Xinje XCPPro project, PLC1: XC2-32 (software 3.3L)

PROGRAM Ladder

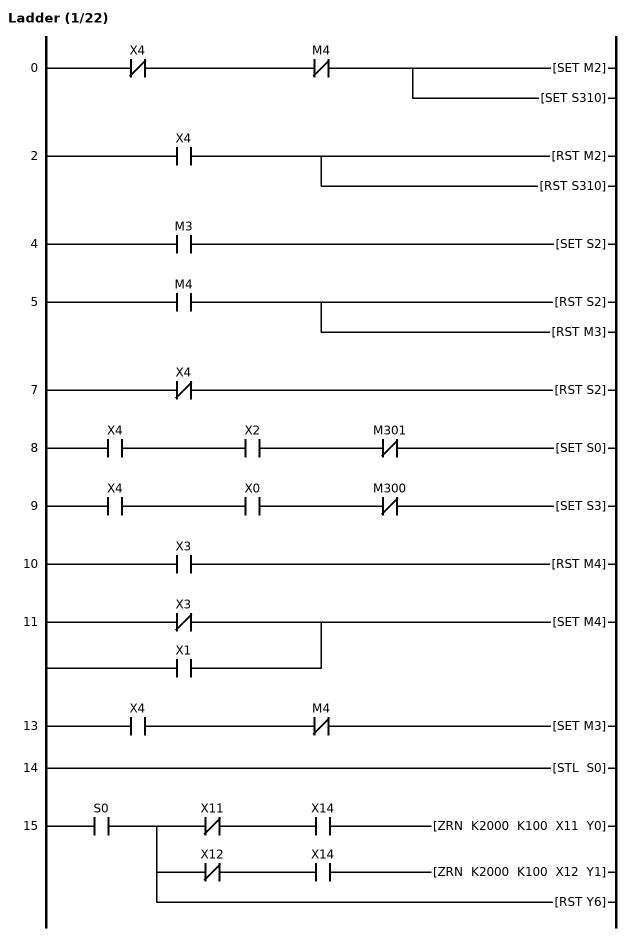
LDI    X4
ANI    M4
SET    M2
SET    S310
LD     X4
RST    M2
RST    S310
LD     M3
SET    S2
LD     M4
RST    S2
RST    M3
LDI    X4
RST    S2
LD     X4
AND    X2
ANI    M301
SET    S0
LD     X4
AND    X0
ANI    M300
SET    S3
LD     X3
RST    M4
LDI    X3
OR     X1
SET    M4
LD     X4
ANI    M4
SET    M3
STL    S0
LD     S0
MPS
ANI    X11
AND    X14
ZRN    K2000 K100 X11 Y0
MRD
ANI    X12
AND    X14
ZRN    K2000 K100 X12 Y1
MPP
RST    Y6

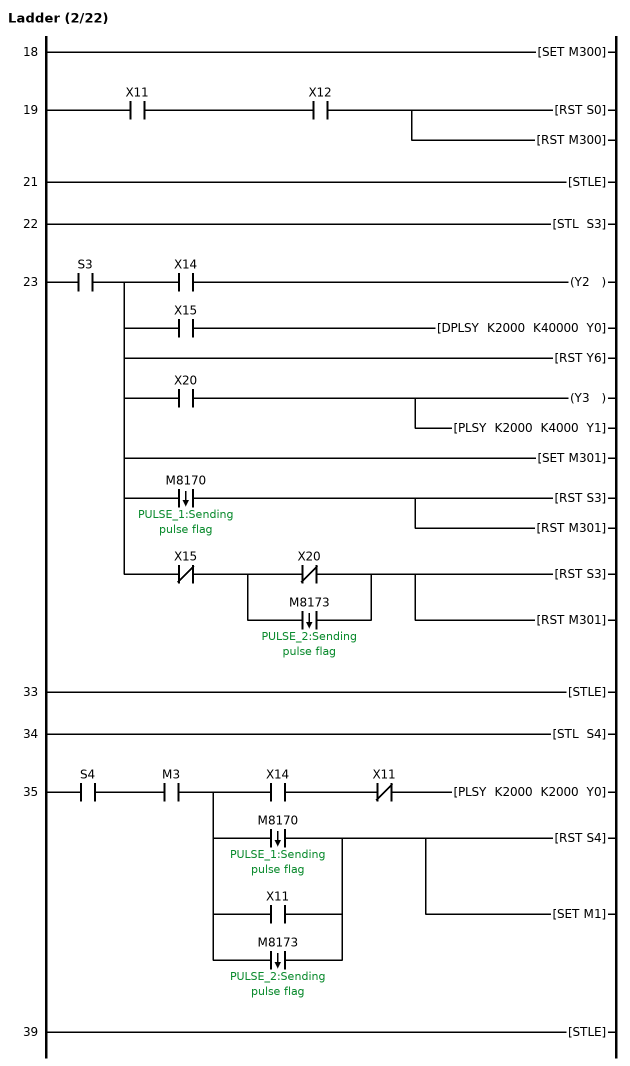
SET    M300
LD     X11
AND    X12
RST    S0
RST    M300
STLE
STL    S3
LD     S3
MPS
AND    X14
OUT    Y2
MRD
AND    X15
DPLSY  K2000 K40000 Y0
MRD
RST    Y6
AND    X20
OUT    Y3
PLSY   K2000 K4000 Y1
MRD
SET    M301
ANDF   M8170	; PULSE_1:Sending pulse flag
RST    S3
RST    M301
MPP
ANI    X15
LDI    X20
ORF    M8173	; PULSE_2:Sending pulse flag
ANB
RST    S3
RST    M301
STLE
STL    S4
LD     S4
AND    M3
MPS
AND    X14
ANI    X11
PLSY   K2000 K2000 Y0
MPP
LDF    M8170	; PULSE_1:Sending pulse flag
OR     X11
ORF    M8173	; PULSE_2:Sending pulse flag
ANB
RST    S4
SET    M1
STLE

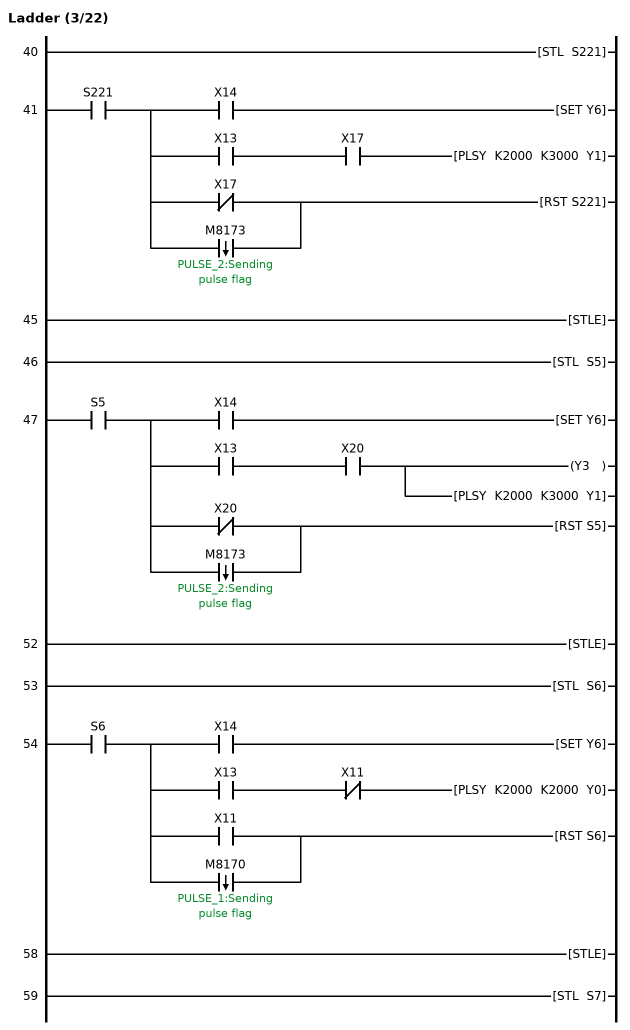
STL    S221
LD     S221
MPS
AND    X14
SET    Y6
MRD
AND    X13
AND    X17
PLSY   K2000 K3000 Y1
MPP
LDI    X17
ORF    M8173	; PULSE_2:Sending pulse flag
ANB
RST    S221
STLE
STL    S5
LD     S5
MPS
AND    X14
SET    Y6
MRD
AND    X13
AND    X20
OUT    Y3
PLSY   K2000 K3000 Y1
MPP
LDI    X20
ORF    M8173	; PULSE_2:Sending pulse flag
ANB
RST    S5
STLE
STL    S6
LD     S6
MPS
AND    X14
SET    Y6
MRD
AND    X13
ANI    X11
PLSY   K2000 K2000 Y0
MPP
LD     X11
ORF    M8170	; PULSE_1:Sending pulse flag
ANB
RST    S6
STLE
STL    S7

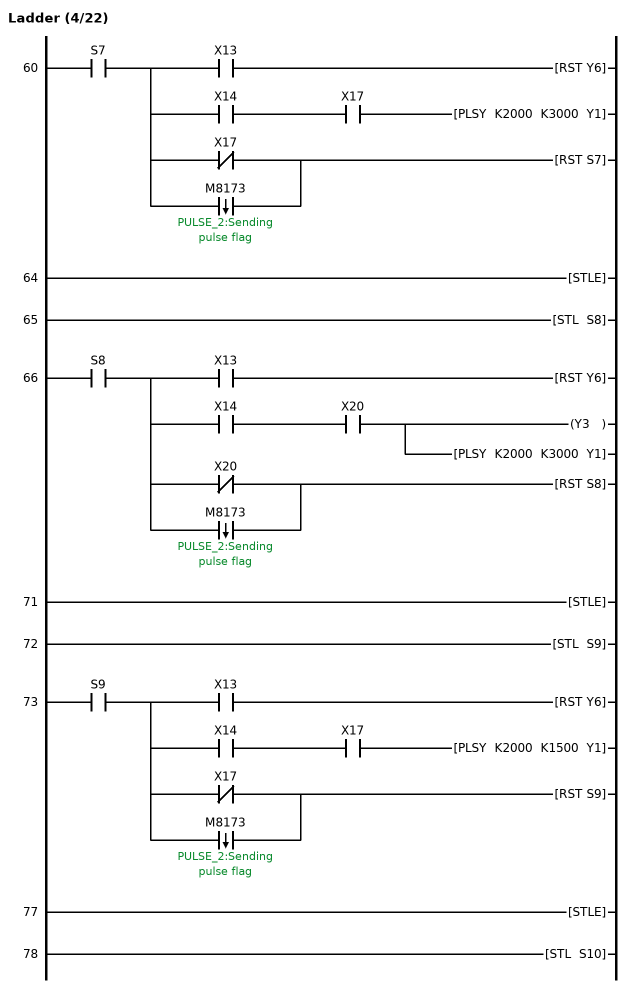
LD     S7
MPS
AND    X13
RST    Y6
MRD
AND    X14
AND    X17
PLSY   K2000 K3000 Y1
MPP
LDI    X17
ORF    M8173	; PULSE_2:Sending pulse flag
ANB
RST    S7
STLE
STL    S8
LD     S8
MPS
AND    X13
RST    Y6
MRD
AND    X14
AND    X20
OUT    Y3
PLSY   K2000 K3000 Y1
MPP
LDI    X20
ORF    M8173	; PULSE_2:Sending pulse flag
ANB
RST    S8
STLE
STL    S9
LD     S9
MPS
AND    X13
RST    Y6
MRD
AND    X14
AND    X17
PLSY   K2000 K1500 Y1
MPP
LDI    X17
ORF    M8173	; PULSE_2:Sending pulse flag
ANB
RST    S9
STLE
STL    S10

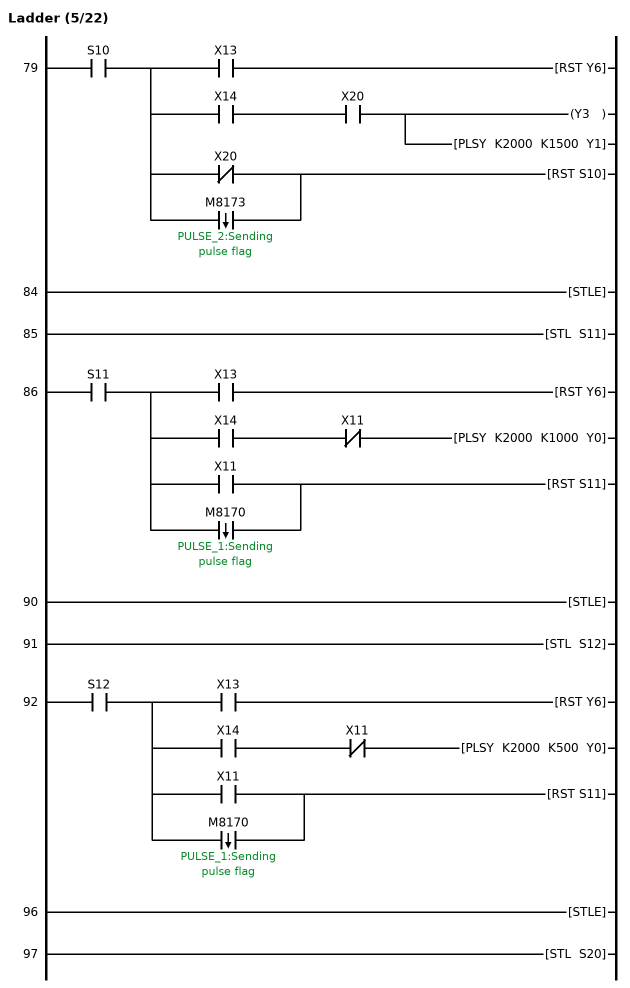
LD     S10
MPS
AND    X13
RST    Y6
MRD
AND    X14
AND    X20
OUT    Y3
PLSY   K2000 K1500 Y1
MPP
LDI    X20
ORF    M8173	; PULSE_2:Sending pulse flag
ANB
RST    S10
STLE
STL    S11
LD     S11
MPS
AND    X13
RST    Y6
MRD
AND    X14
ANI    X11
PLSY   K2000 K1000 Y0
MPP
LD     X11
ORF    M8170	; PULSE_1:Sending pulse flag
ANB
RST    S11
STLE
STL    S12
LD     S12
MPS
AND    X13
RST    Y6
MRD
AND    X14
ANI    X11
PLSY   K2000 K500 Y0
MPP
LD     X11
ORF    M8170	; PULSE_1:Sending pulse flag
ANB
RST    S11
STLE
STL    S20

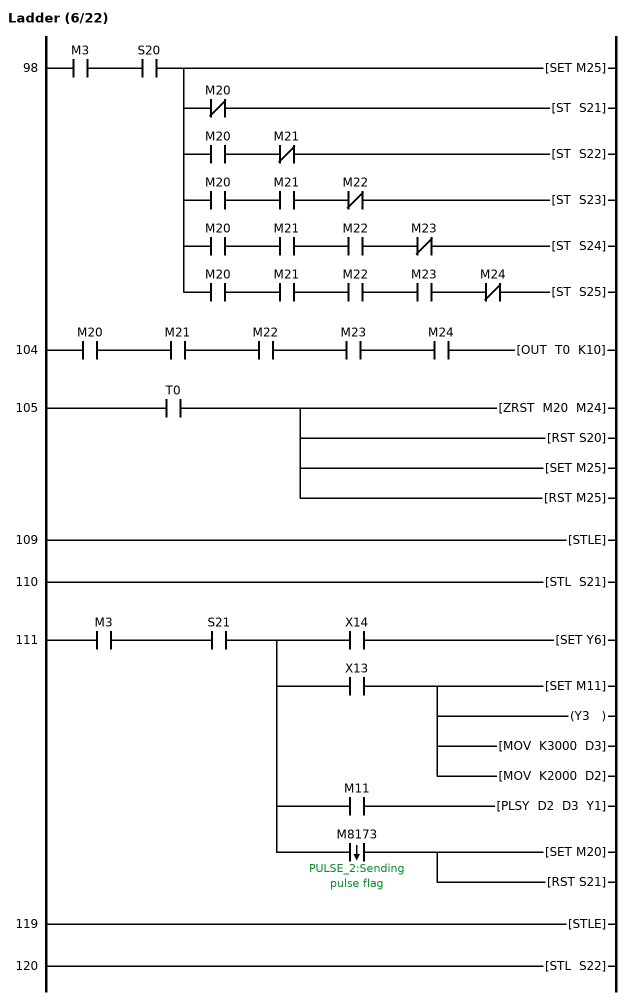
LD     M3
AND    S20
SET    M25
MPS
ANI    M20
ST     S21
MRD
AND    M20
ANI    M21
ST     S22
MRD
AND    M20
AND    M21
ANI    M22
ST     S23
MRD
AND    M20
AND    M21
AND    M22
ANI    M23
ST     S24
MPP
AND    M20
AND    M21
AND    M22
AND    M23
ANI    M24
ST     S25
LD     M20
AND    M21
AND    M22
AND    M23
AND    M24
OUT    T0 K10
LD     T0
ZRST   M20 M24
RST    S20
SET    M25
RST    M25
STLE
STL    S21
LD     M3
AND    S21
MPS
AND    X14
SET    Y6
MRD
AND    X13
SET    M11
OUT    Y3
MOV    K3000 D3
MOV    K2000 D2
MRD
AND    M11
PLSY   D2 D3 Y1
MPP
ANDF   M8173	; PULSE_2:Sending pulse flag
SET    M20
RST    S21
STLE
STL    S22

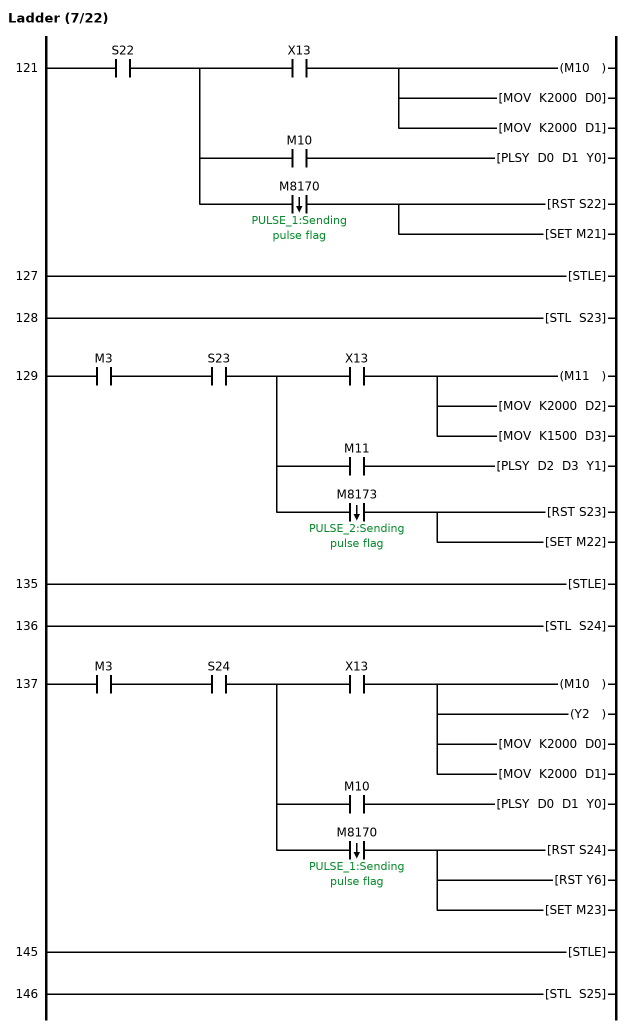
LD     S22
MPS
AND    X13
OUT    M10
MOV    K2000 D0
MOV    K2000 D1
MRD
AND    M10
PLSY   D0 D1 Y0
MPP
ANDF   M8170	; PULSE_1:Sending pulse flag
RST    S22
SET    M21
STLE
STL    S23
LD     M3
AND    S23
MPS
AND    X13
OUT    M11
MOV    K2000 D2
MOV    K1500 D3
MRD
AND    M11
PLSY   D2 D3 Y1
MPP
ANDF   M8173	; PULSE_2:Sending pulse flag
RST    S23
SET    M22
STLE
STL    S24
LD     M3
AND    S24
MPS
AND    X13
OUT    M10
OUT    Y2
MOV    K2000 D0
MOV    K2000 D1
MRD
AND    M10
PLSY   D0 D1 Y0
MPP
ANDF   M8170	; PULSE_1:Sending pulse flag
RST    S24
RST    Y6
SET    M23
STLE
STL    S25

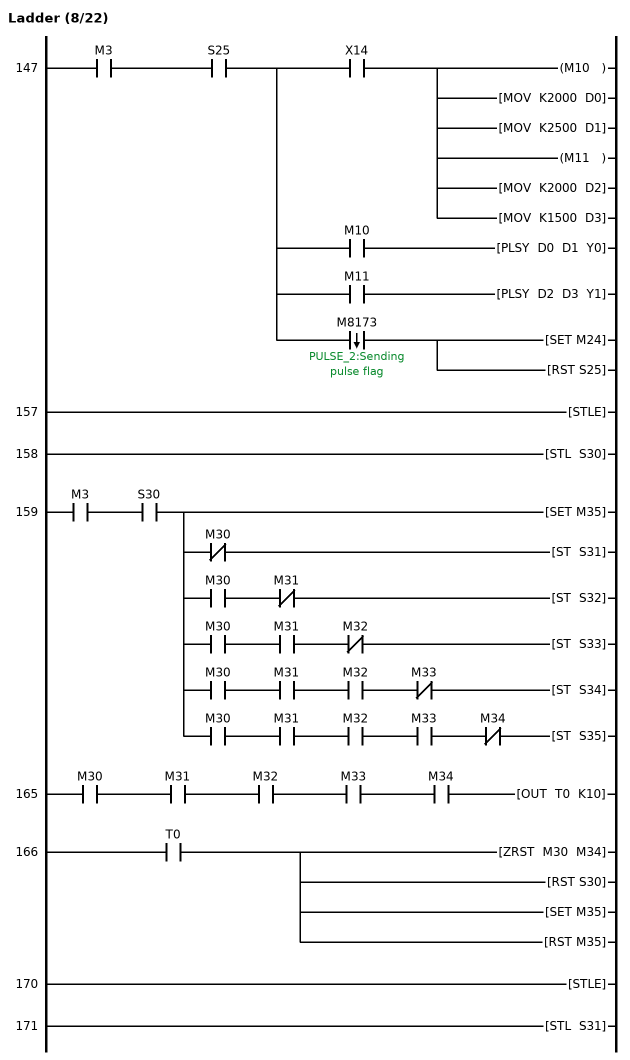
LD     M3
AND    S25
MPS
AND    X14
OUT    M10
MOV    K2000 D0
MOV    K2500 D1
OUT    M11
MOV    K2000 D2
MOV    K1500 D3
MRD
AND    M10
PLSY   D0 D1 Y0
MRD
AND    M11
PLSY   D2 D3 Y1
MPP
ANDF   M8173	; PULSE_2:Sending pulse flag
SET    M24
RST    S25
STLE
STL    S30
LD     M3
AND    S30
SET    M35
MPS
ANI    M30
ST     S31
MRD
AND    M30
ANI    M31
ST     S32
MRD
AND    M30
AND    M31
ANI    M32
ST     S33
MRD
AND    M30
AND    M31
AND    M32
ANI    M33
ST     S34
MPP
AND    M30
AND    M31
AND    M32
AND    M33
ANI    M34
ST     S35
LD     M30
AND    M31
AND    M32
AND    M33
AND    M34
OUT    T0 K10
LD     T0
ZRST   M30 M34
RST    S30
SET    M35
RST    M35
STLE
STL    S31

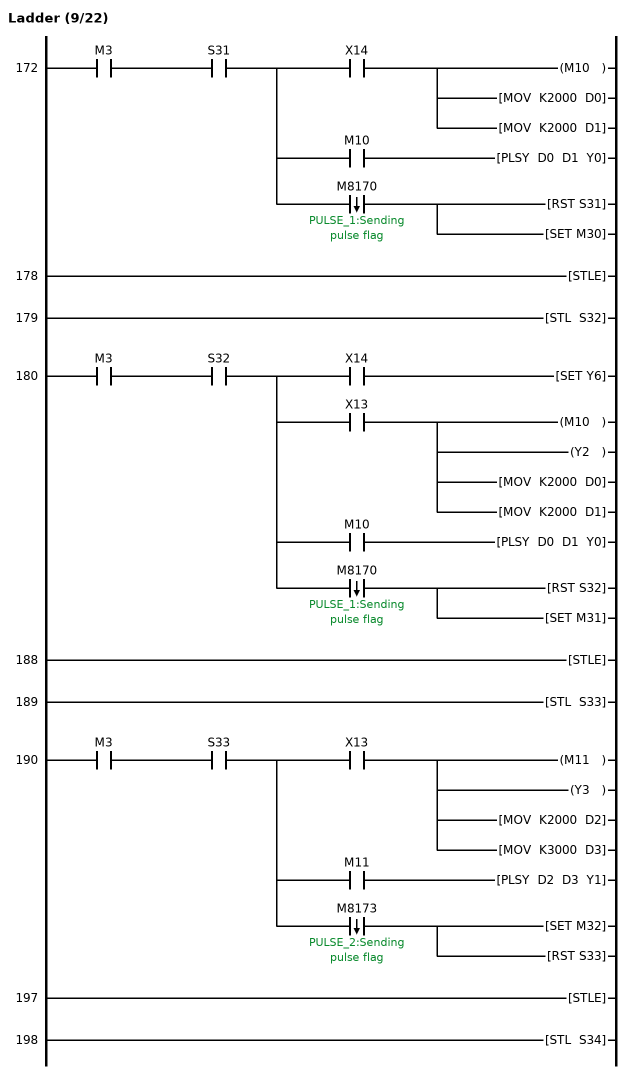
LD     M3
AND    S31
MPS
AND    X14
OUT    M10
MOV    K2000 D0
MOV    K2000 D1
MRD
AND    M10
PLSY   D0 D1 Y0
MPP
ANDF   M8170	; PULSE_1:Sending pulse flag
RST    S31
SET    M30
STLE
STL    S32
LD     M3
AND    S32
MPS
AND    X14
SET    Y6
MRD
AND    X13
OUT    M10
OUT    Y2
MOV    K2000 D0
MOV    K2000 D1
MRD
AND    M10
PLSY   D0 D1 Y0
MPP
ANDF   M8170	; PULSE_1:Sending pulse flag
RST    S32
SET    M31
STLE
STL    S33
LD     M3
AND    S33
MPS
AND    X13
OUT    M11
OUT    Y3
MOV    K2000 D2
MOV    K3000 D3
MRD
AND    M11
PLSY   D2 D3 Y1
MPP
ANDF   M8173	; PULSE_2:Sending pulse flag
SET    M32
RST    S33
STLE
STL    S34

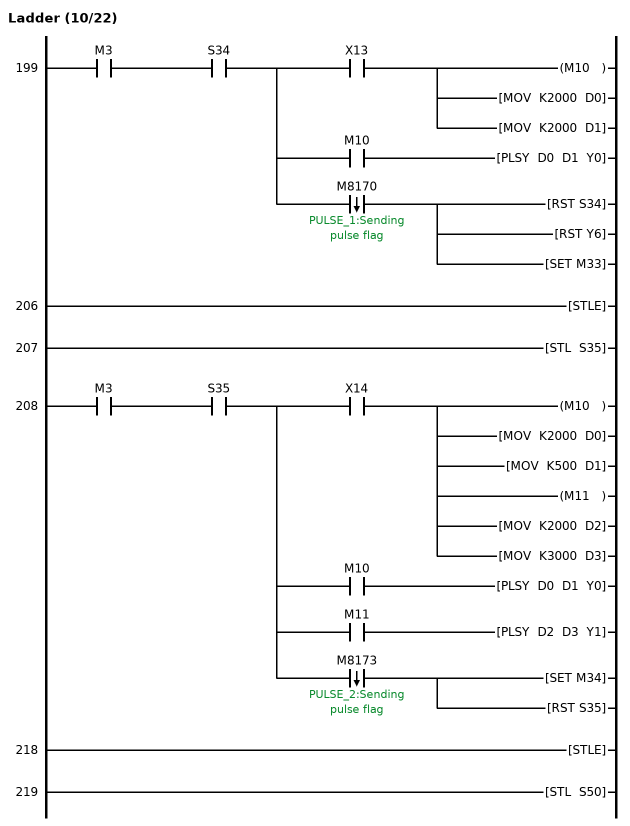
LD     M3
AND    S34
MPS
AND    X13
OUT    M10
MOV    K2000 D0
MOV    K2000 D1
MRD
AND    M10
PLSY   D0 D1 Y0
MPP
ANDF   M8170	; PULSE_1:Sending pulse flag
RST    S34
RST    Y6
SET    M33
STLE
STL    S35
LD     M3
AND    S35
MPS
AND    X14
OUT    M10
MOV    K2000 D0
MOV    K500 D1
OUT    M11
MOV    K2000 D2
MOV    K3000 D3
MRD
AND    M10
PLSY   D0 D1 Y0
MRD
AND    M11
PLSY   D2 D3 Y1
MPP
ANDF   M8173	; PULSE_2:Sending pulse flag
SET    M34
RST    S35
STLE
STL    S50

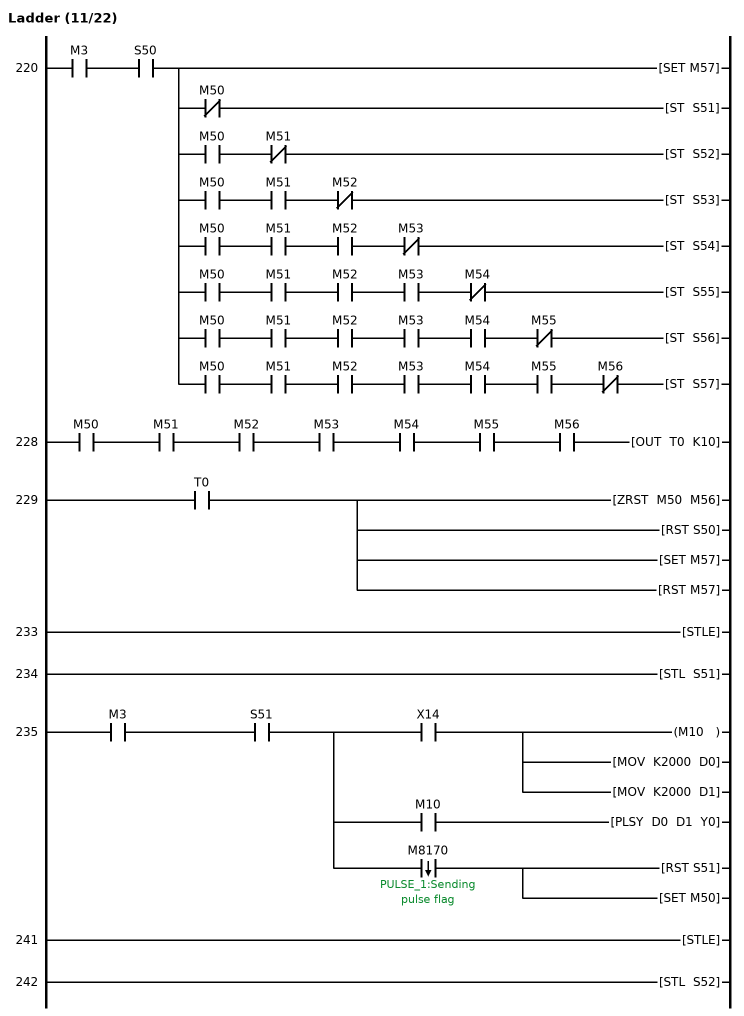
LD     M3
AND    S50
SET    M57
MPS
ANI    M50
ST     S51
MRD
AND    M50
ANI    M51
ST     S52
MRD
AND    M50
AND    M51
ANI    M52
ST     S53
MRD
AND    M50
AND    M51
AND    M52
ANI    M53
ST     S54
MRD
AND    M50
AND    M51
AND    M52
AND    M53
ANI    M54
ST     S55
MRD
AND    M50
AND    M51
AND    M52
AND    M53
AND    M54
ANI    M55
ST     S56
MPP
AND    M50
AND    M51
AND    M52
AND    M53
AND    M54
AND    M55
ANI    M56
ST     S57
LD     M50
AND    M51
AND    M52
AND    M53
AND    M54
AND    M55
AND    M56
OUT    T0 K10
LD     T0
ZRST   M50 M56
RST    S50
SET    M57
RST    M57
STLE
STL    S51
LD     M3
AND    S51
MPS
AND    X14
OUT    M10
MOV    K2000 D0
MOV    K2000 D1
MRD
AND    M10
PLSY   D0 D1 Y0
MPP
ANDF   M8170	; PULSE_1:Sending pulse flag
RST    S51
SET    M50
STLE
STL    S52

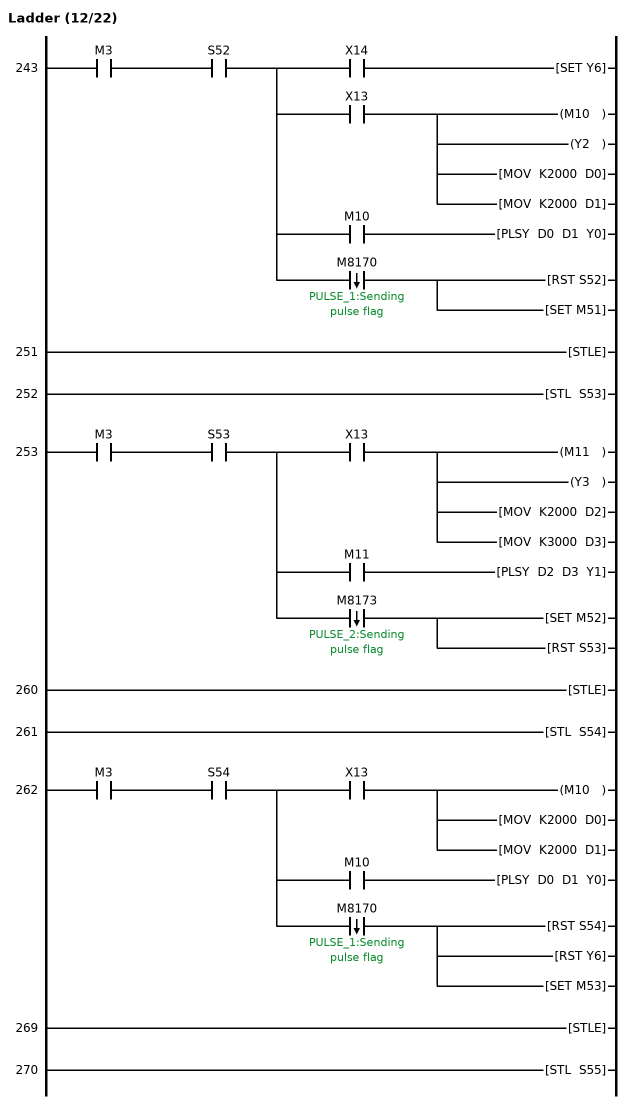
LD     M3
AND    S52
MPS
AND    X14
SET    Y6
MRD
AND    X13
OUT    M10
OUT    Y2
MOV    K2000 D0
MOV    K2000 D1
MRD
AND    M10
PLSY   D0 D1 Y0
MPP
ANDF   M8170	; PULSE_1:Sending pulse flag
RST    S52
SET    M51
STLE
STL    S53
LD     M3
AND    S53
MPS
AND    X13
OUT    M11
OUT    Y3
MOV    K2000 D2
MOV    K3000 D3
MRD
AND    M11
PLSY   D2 D3 Y1
MPP
ANDF   M8173	; PULSE_2:Sending pulse flag
SET    M52
RST    S53
STLE
STL    S54
LD     M3
AND    S54
MPS
AND    X13
OUT    M10
MOV    K2000 D0
MOV    K2000 D1
MRD
AND    M10
PLSY   D0 D1 Y0
MPP
ANDF   M8170	; PULSE_1:Sending pulse flag
RST    S54
RST    Y6
SET    M53
STLE
STL    S55

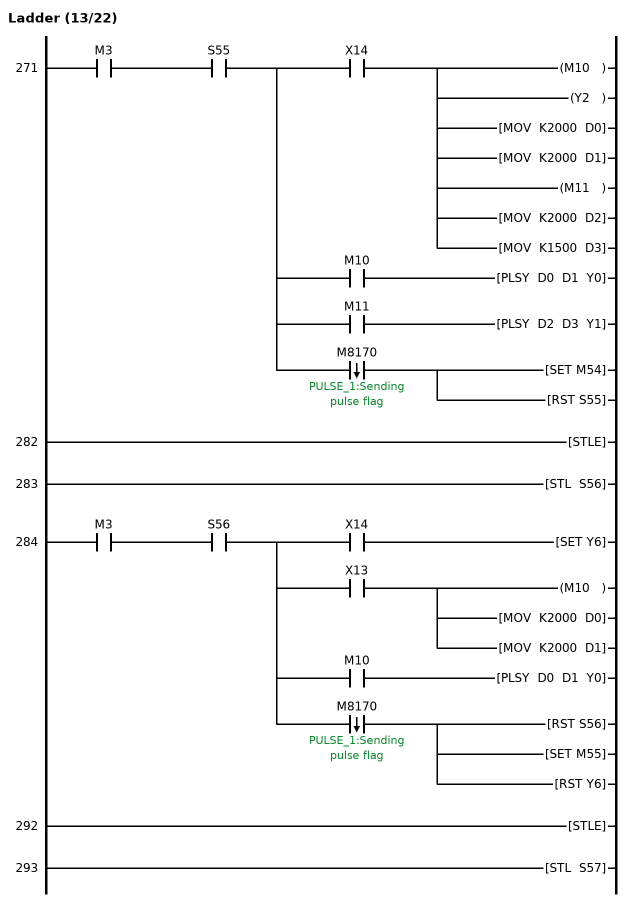
LD     M3
AND    S55
MPS
AND    X14
OUT    M10
OUT    Y2
MOV    K2000 D0
MOV    K2000 D1
OUT    M11
MOV    K2000 D2
MOV    K1500 D3
MRD
AND    M10
PLSY   D0 D1 Y0
MRD
AND    M11
PLSY   D2 D3 Y1
MPP
ANDF   M8170	; PULSE_1:Sending pulse flag
SET    M54
RST    S55
STLE
STL    S56
LD     M3
AND    S56
MPS
AND    X14
SET    Y6
MRD
AND    X13
OUT    M10
MOV    K2000 D0
MOV    K2000 D1
MRD
AND    M10
PLSY   D0 D1 Y0
MPP
ANDF   M8170	; PULSE_1:Sending pulse flag
RST    S56
SET    M55
RST    Y6
STLE
STL    S57

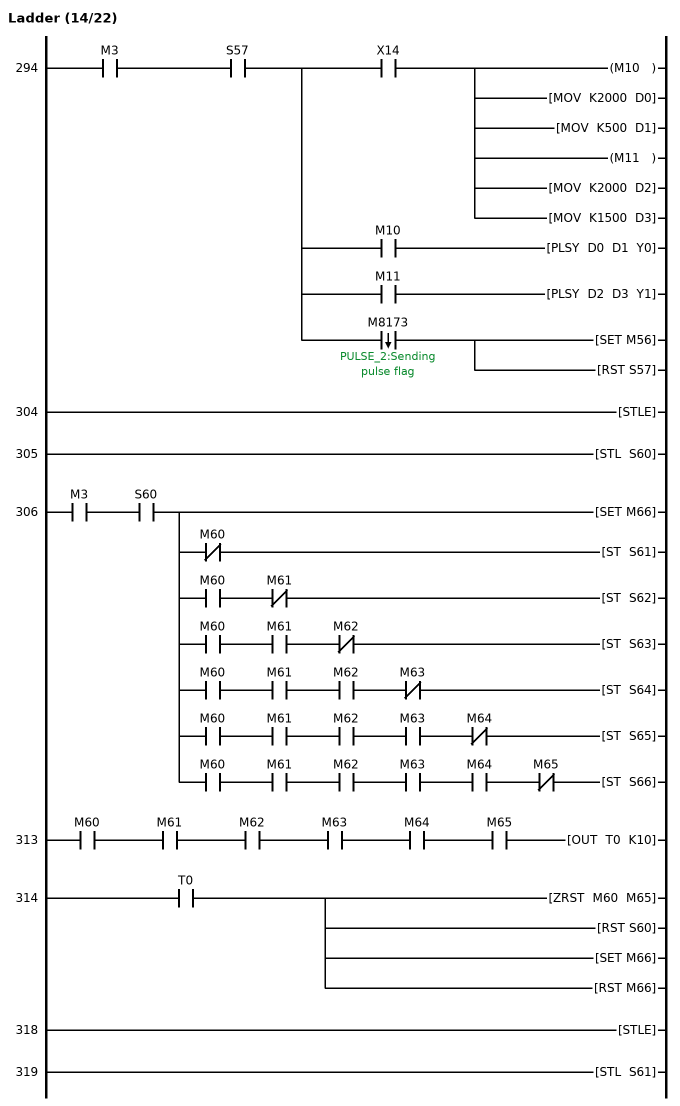
LD     M3
AND    S57
MPS
AND    X14
OUT    M10
MOV    K2000 D0
MOV    K500 D1
OUT    M11
MOV    K2000 D2
MOV    K1500 D3
MRD
AND    M10
PLSY   D0 D1 Y0
MRD
AND    M11
PLSY   D2 D3 Y1
MPP
ANDF   M8173	; PULSE_2:Sending pulse flag
SET    M56
RST    S57
STLE
STL    S60
LD     M3
AND    S60
SET    M66
MPS
ANI    M60
ST     S61
MRD
AND    M60
ANI    M61
ST     S62
MRD
AND    M60
AND    M61
ANI    M62
ST     S63
MRD
AND    M60
AND    M61
AND    M62
ANI    M63
ST     S64
MRD
AND    M60
AND    M61
AND    M62
AND    M63
ANI    M64
ST     S65
MPP
AND    M60
AND    M61
AND    M62
AND    M63
AND    M64
ANI    M65
ST     S66
LD     M60
AND    M61
AND    M62
AND    M63
AND    M64
AND    M65
OUT    T0 K10
LD     T0
ZRST   M60 M65
RST    S60
SET    M66
RST    M66
STLE
STL    S61

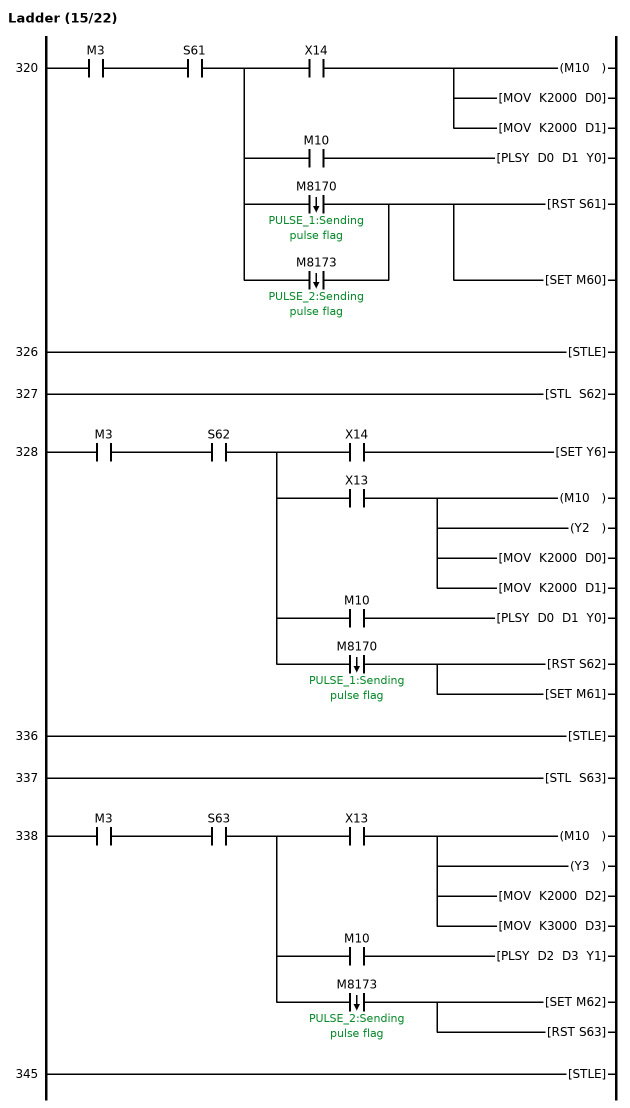
LD     M3
AND    S61
MPS
AND    X14
OUT    M10
MOV    K2000 D0
MOV    K2000 D1
MRD
AND    M10
PLSY   D0 D1 Y0
MPP
LDF    M8170	; PULSE_1:Sending pulse flag
ORF    M8173	; PULSE_2:Sending pulse flag
ANB
RST    S61
SET    M60
STLE
STL    S62
LD     M3
AND    S62
MPS
AND    X14
SET    Y6
MRD
AND    X13
OUT    M10
OUT    Y2
MOV    K2000 D0
MOV    K2000 D1
MRD
AND    M10
PLSY   D0 D1 Y0
MPP
ANDF   M8170	; PULSE_1:Sending pulse flag
RST    S62
SET    M61
STLE
STL    S63
LD     M3
AND    S63
MPS
AND    X13
OUT    M10
OUT    Y3
MOV    K2000 D2
MOV    K3000 D3
MRD
AND    M10
PLSY   D2 D3 Y1
MPP
ANDF   M8173	; PULSE_2:Sending pulse flag
SET    M62
RST    S63
STLE

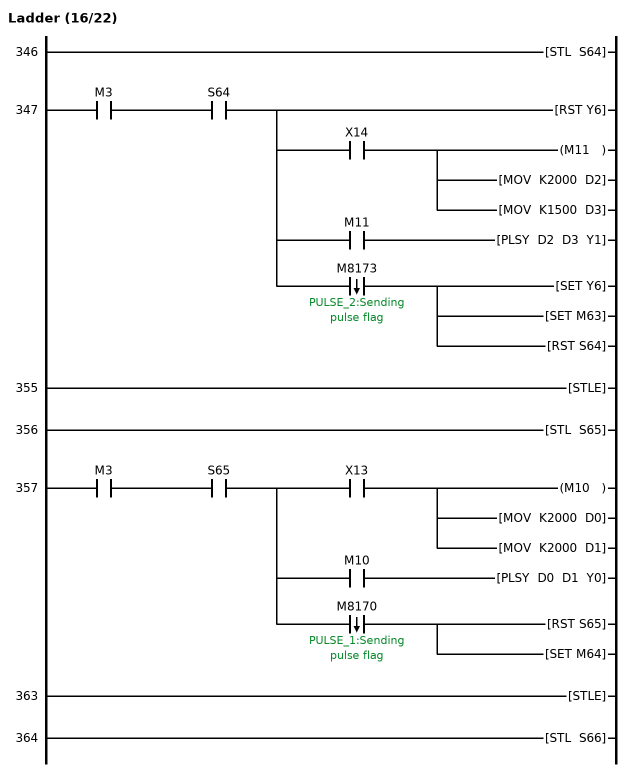
STL    S64
LD     M3
AND    S64
RST    Y6
MPS
AND    X14
OUT    M11
MOV    K2000 D2
MOV    K1500 D3
MRD
AND    M11
PLSY   D2 D3 Y1
MPP
ANDF   M8173	; PULSE_2:Sending pulse flag
SET    Y6
SET    M63
RST    S64
STLE
STL    S65
LD     M3
AND    S65
MPS
AND    X13
OUT    M10
MOV    K2000 D0
MOV    K2000 D1
MRD
AND    M10
PLSY   D0 D1 Y0
MPP
ANDF   M8170	; PULSE_1:Sending pulse flag
RST    S65
SET    M64
STLE
STL    S66

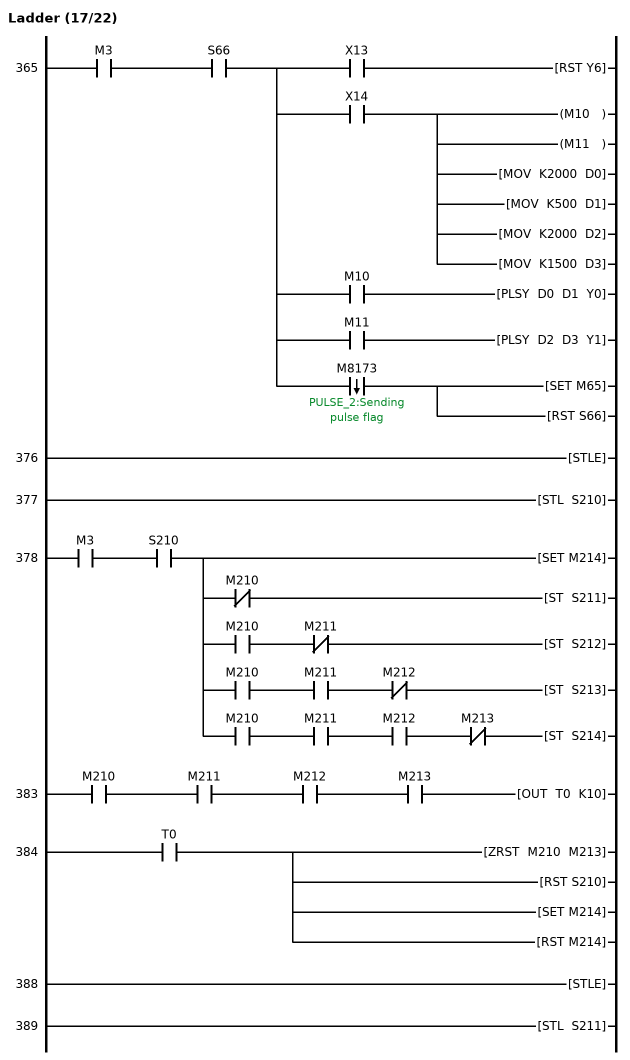
LD     M3
AND    S66
MPS
AND    X13
RST    Y6
MRD
AND    X14
OUT    M10
OUT    M11
MOV    K2000 D0
MOV    K500 D1
MOV    K2000 D2
MOV    K1500 D3
MRD
AND    M10
PLSY   D0 D1 Y0
MRD
AND    M11
PLSY   D2 D3 Y1
MPP
ANDF   M8173	; PULSE_2:Sending pulse flag
SET    M65
RST    S66
STLE
STL    S210
LD     M3
AND    S210
SET    M214
MPS
ANI    M210
ST     S211
MRD
AND    M210
ANI    M211
ST     S212
MRD
AND    M210
AND    M211
ANI    M212
ST     S213
MPP
AND    M210
AND    M211
AND    M212
ANI    M213
ST     S214
LD     M210
AND    M211
AND    M212
AND    M213
OUT    T0 K10
LD     T0
ZRST   M210 M213
RST    S210
SET    M214
RST    M214
STLE
STL    S211

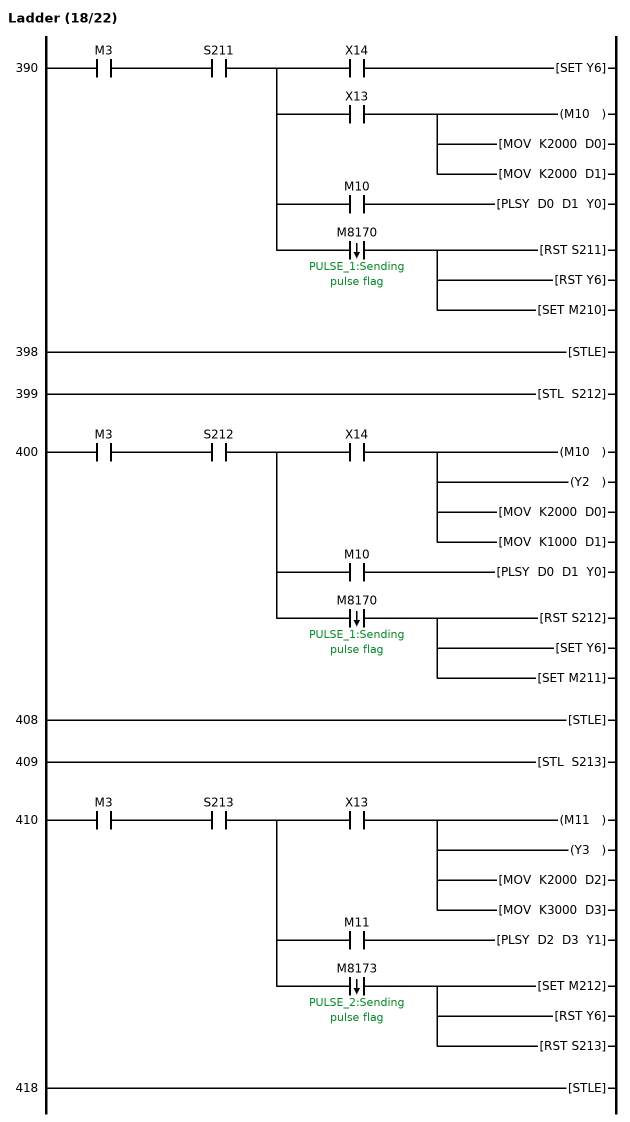
LD     M3
AND    S211
MPS
AND    X14
SET    Y6
MRD
AND    X13
OUT    M10
MOV    K2000 D0
MOV    K2000 D1
MRD
AND    M10
PLSY   D0 D1 Y0
MPP
ANDF   M8170	; PULSE_1:Sending pulse flag
RST    S211
RST    Y6
SET    M210
STLE
STL    S212
LD     M3
AND    S212
MPS
AND    X14
OUT    M10
OUT    Y2
MOV    K2000 D0
MOV    K1000 D1
MRD
AND    M10
PLSY   D0 D1 Y0
MPP
ANDF   M8170	; PULSE_1:Sending pulse flag
RST    S212
SET    Y6
SET    M211
STLE
STL    S213
LD     M3
AND    S213
MPS
AND    X13
OUT    M11
OUT    Y3
MOV    K2000 D2
MOV    K3000 D3
MRD
AND    M11
PLSY   D2 D3 Y1
MPP
ANDF   M8173	; PULSE_2:Sending pulse flag
SET    M212
RST    Y6
RST    S213
STLE

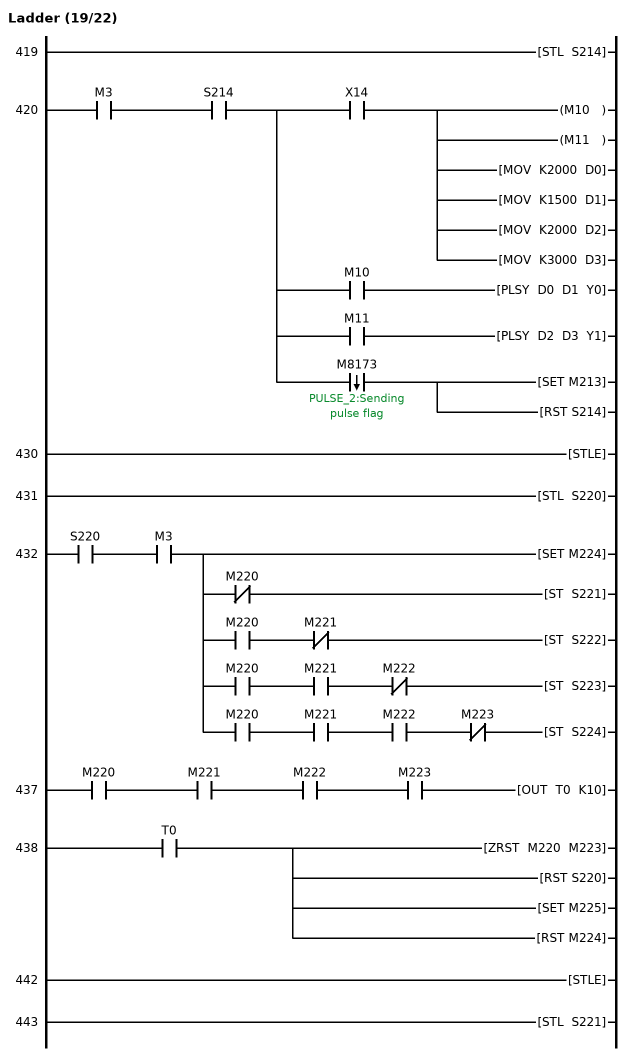
STL    S214
LD     M3
AND    S214
MPS
AND    X14
OUT    M10
OUT    M11
MOV    K2000 D0
MOV    K1500 D1
MOV    K2000 D2
MOV    K3000 D3
MRD
AND    M10
PLSY   D0 D1 Y0
MRD
AND    M11
PLSY   D2 D3 Y1
MPP
ANDF   M8173	; PULSE_2:Sending pulse flag
SET    M213
RST    S214
STLE
STL    S220
LD     S220
AND    M3
SET    M224
MPS
ANI    M220
ST     S221
MRD
AND    M220
ANI    M221
ST     S222
MRD
AND    M220
AND    M221
ANI    M222
ST     S223
MPP
AND    M220
AND    M221
AND    M222
ANI    M223
ST     S224
LD     M220
AND    M221
AND    M222
AND    M223
OUT    T0 K10
LD     T0
ZRST   M220 M223
RST    S220
SET    M225
RST    M224
STLE
STL    S221

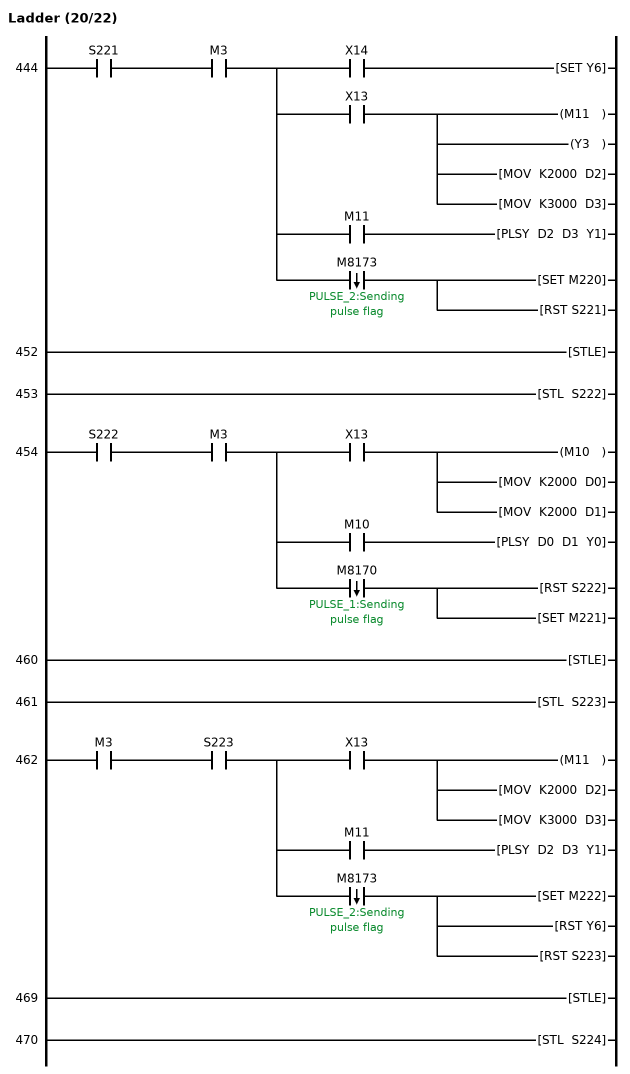
LD     S221
AND    M3
MPS
AND    X14
SET    Y6
MRD
AND    X13
OUT    M11
OUT    Y3
MOV    K2000 D2
MOV    K3000 D3
MRD
AND    M11
PLSY   D2 D3 Y1
MPP
ANDF   M8173	; PULSE_2:Sending pulse flag
SET    M220
RST    S221
STLE
STL    S222
LD     S222
AND    M3
MPS
AND    X13
OUT    M10
MOV    K2000 D0
MOV    K2000 D1
MRD
AND    M10
PLSY   D0 D1 Y0
MPP
ANDF   M8170	; PULSE_1:Sending pulse flag
RST    S222
SET    M221
STLE
STL    S223
LD     M3
AND    S223
MPS
AND    X13
OUT    M11
MOV    K2000 D2
MOV    K3000 D3
MRD
AND    M11
PLSY   D2 D3 Y1
MPP
ANDF   M8173	; PULSE_2:Sending pulse flag
SET    M222
RST    Y6
RST    S223
STLE
STL    S224

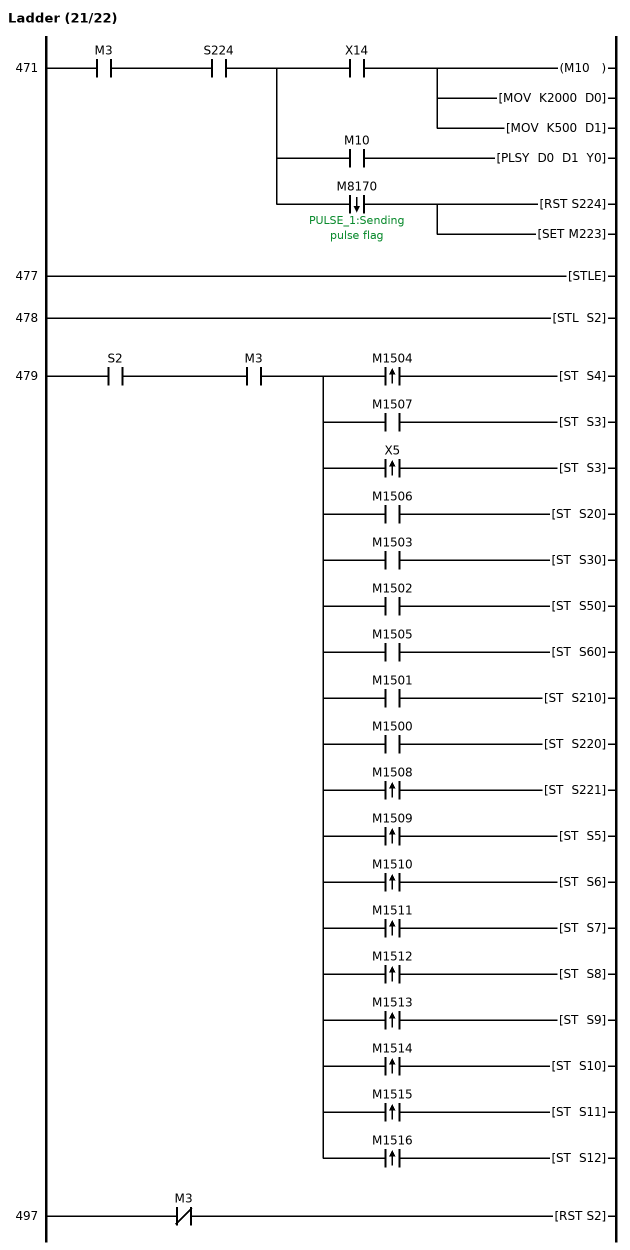
LD     M3
AND    S224
MPS
AND    X14
OUT    M10
MOV    K2000 D0
MOV    K500 D1
MRD
AND    M10
PLSY   D0 D1 Y0
MPP
ANDF   M8170	; PULSE_1:Sending pulse flag
RST    S224
SET    M223
STLE
STL    S2
LD     S2
AND    M3
MPS
ANDP   M1504
ST     S4
MRD
AND    M1507
ST     S3
MRD
ANDP   X5
ST     S3
MRD
AND    M1506
ST     S20
MRD
AND    M1503
ST     S30
MRD
AND    M1502
ST     S50
MRD
AND    M1505
ST     S60
MRD
AND    M1501
ST     S210
MRD
AND    M1500
ST     S220
MRD
ANDP   M1508
ST     S221
MRD
ANDP   M1509
ST     S5
MRD
ANDP   M1510
ST     S6
MRD
ANDP   M1511
ST     S7
MRD
ANDP   M1512
ST     S8
MRD
ANDP   M1513
ST     S9
MRD
ANDP   M1514
ST     S10
MRD
ANDP   M1515
ST     S11
MPP
ANDP   M1516
ST     S12
LDI    M3
RST    S2

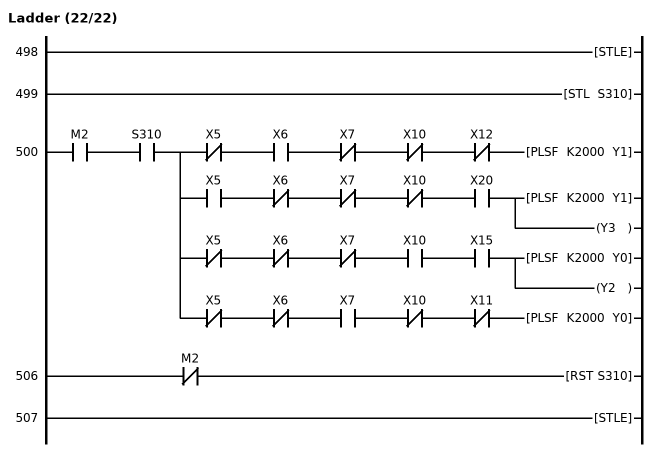
STLE
STL    S310
LD     M2
AND    S310
MPS
ANI    X5
AND    X6
ANI    X7
ANI    X10
ANI    X12
PLSF   K2000 Y1
MRD
AND    X5
ANI    X6
ANI    X7
ANI    X10
AND    X20
PLSF   K2000 Y1
OUT    Y3
MRD
ANI    X5
ANI    X6
ANI    X7
AND    X10
AND    X15
PLSF   K2000 Y0
OUT    Y2
MPP
ANI    X5
ANI    X6
AND    X7
ANI    X10
ANI    X11
PLSF   K2000 Y0
LDI    M2
RST    S310
STLE